RESOURCE_TYPE _Core
  (* Standard: 61499-2 *)
  (* Version 0.1, 2017-00-02, hpea485, UOA *)
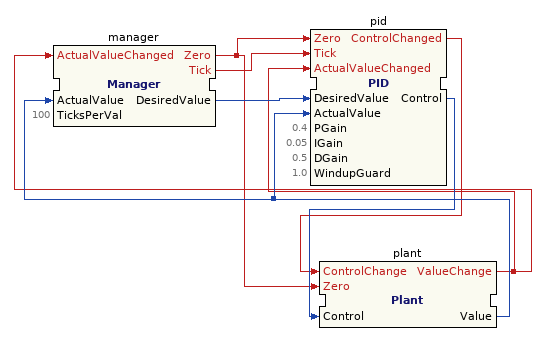
  FBS
    pid : PID(PGain := 0.4, IGain := 0.05, DGain := 0.5, WindupGuard := 1.0);
    manager : Manager(TicksPerVal := 100);
    plant : Plant;
  END_FBS
  EVENT_CONNECTIONS
    pid.ControlChanged TO plant.ControlChange;
    manager.Zero TO pid.Zero;
    manager.Zero TO plant.Zero;
    manager.Tick TO pid.Tick;
    plant.ValueChange TO manager.ActualValueChanged;
    plant.ValueChange TO pid.ActualValueChanged;
  END_CONNECTIONS
  DATA_CONNECTIONS
    pid.Control TO plant.Control;
    manager.DesiredValue TO pid.DesiredValue;
    plant.Value TO pid.ActualValue;
    plant.Value TO manager.ActualValue;
  END_CONNECTIONS
END_RESOURCE_TYPE
